// TIA Portal project "analog_kanaldan_alinan_degeri_skala _etme" (V18)

(* hardware
DEVICE "S7-1200 station_1"  S7-1200 Station
   slot 0: "Rack_0"  S7-1200 Rack  Rack  V1.0
   slot 1: "PLC_1"  CPU 1214C AC/DC/Rly  6ES7 214-1BG40-0XB0  V4.6
*)

// ===== PLC "PLC_1"  CPU 1214C AC/DC/Rly =====

VAR_GLOBAL   // PLC tag table "Default tag table"
   "Tag_1" AT %IW64 : Word;
   "Tag_2" AT %MD70 : DWord;
   "Tag_3" AT %MD80 : Real;
   "Tag_4" AT %MW60 : Int;
END_VAR

ORGANIZATION_BLOCK "Main"   // OB1, LAD, ProgramCycle
TITLE = "Main Program Sweep (Cycle)"
{ S7_Optimized_Access := 'TRUE' }
VERSION : 0.1
   VAR_INPUT
      Initial_Call : Bool;   // Initial call of this OB
      Remanence : Bool;   // =True, if remanent data are available
   END_VAR
BEGIN

REGION Network 1
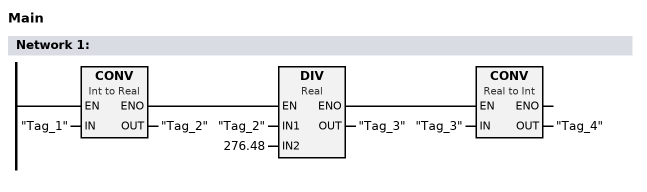
   RUNG wire#powerrail
      { S7_Templates := "[SrcType := Int, DestType := Real]" } Convert(in := "Tag_1", out => "Tag_2")
      { S7_Templates := "SrcType := Real" } Div(in1 := "Tag_2", in2 := 276.48, out => "Tag_3")
      { S7_Templates := "[SrcType := Real, DestType := Int]" } Convert(in := "Tag_3", out => "Tag_4")
   END_RUNG
   // the same network as SCL:
   "Tag_2" := INT_TO_REAL("Tag_1");
   "Tag_3" := "Tag_2" / 276.48;
   "Tag_4" := REAL_TO_INT("Tag_3");
END_REGION
END_ORGANIZATION_BLOCK